FUNCTION_BLOCK FB_QM_MinDirChanges IMPLEMENTS IF_queueManager
VAR_INPUT
	bButtons 	  : ARRAY [1..NUMLEVELS] OF BOOL;						(* user input *)
END_VAR
VAR_OUTPUT
END_VAR
VAR
	tPushDetects  : ARRAY [1..NUMLEVELS] OF FB_BinaryInp;				(* FBs to buffer user inputs until being processed *)
	queueManip	  : FB_ArrManip;										(* FB for array manipulation, like sorting etc. *)
	k			  : INT;												(* loop variable *)
	eDirection    : LiftMovingDirection := LiftMovingDirection.up;		(* local variable for moving direction *)
	
	nCurLevel	  : INT(1..NUMLEVELS);									(* current lift position *)
	nQueue		  : ARRAY [1..NUMLEVELS] OF INT;						(* queue, saving next targets in current moving direction *)
	bLevelInQueue : ARRAY [1..NUMLEVELS] OF BOOL;						(* buffer of all active calls , i.e. levels in nQueue OR active tPushDetects *)
END_VAR

FOR k:=1 TO NUMLEVELS DO
	tPushDetects[k](bPush:=bButtons[k], bReset:=FALSE);
	bLevelInQueue[k] := tPushDetects[k].bOutActive OR queueManip.isElement(arr:=nQueue, entry:=k);
END_FOR

FOR k:=1 TO NUMLEVELS DO
	IF tPushDetects[k].bOutActive THEN
		IF queueManip.isEmpty(arr:=nQueue, emptyElement:=0) THEN
			// Queue is empty. Just inset new element and sort desc (-> new Element is at front)
			queueManip.insert(arr:=nQueue, newElement:=k, freeElement:=0);
			queueManip.quicksort_desc(arr:=nQueue, lo:=1, hi:=NUMLEVELS);
			// ... and set Direction to UP if current lift position is below the calling level
			IF nCurLevel < k THEN
				eDirection := LiftMovingDirection.up;
			END_IF
			// ... and set Direction to DOWN if current lift position is above the calling level
			IF nCurLevel > k THEN
				eDirection := LiftMovingDirection.down;
			END_IF
			// otherwise leave direction as it is!
			
			// Then acknowledge
			tPushDetects[k](bReset:=TRUE);
			CONTINUE;
		END_IF	
	
		(*
			if new call is already included in queue, then acknowldge
			and continue with next loop iteration 
		*)
		IF queueManip.isElement(arr:=nQueue, entry:=k) THEN
			tPushDetects[k](bReset:=TRUE);
			CONTINUE;
		END_IF
		
		(* 
			lift is moving up and new call is from above the lift position,
			so the new call in inserted into queue and queue is sorted afterwards.
		*)
		IF nCurLevel < k AND eDirection = LiftMovingDirection.up THEN
			queueManip.insert(arr:=nQueue, newElement:=k, freeElement:=0);
			queueManip.quicksort_asc(arr:=nQueue, lo:=1, hi:=NUMLEVELS);
			WHILE nQueue[1] = 0 DO
				queueManip.pop_front(arr:=nQueue, fill:=0);
			END_WHILE
			// ack call
			tPushDetects[k](bReset:=TRUE);
		END_IF
		
		(* 
			lift is moving down and new call is from below the lift position,
			so the new call in inserted into queue and queue is sorted afterwards.
		*)
		IF nCurLevel > k AND eDirection = LiftMovingDirection.down THEN
			queueManip.insert(arr:=nQueue, newElement:=k, freeElement:=0);
			queueManip.quicksort_desc(arr:=nQueue, lo:=1, hi:=NUMLEVELS);
			// ack call
			tPushDetects[k](bReset:=TRUE);
		END_IF
	END_IF
END_FOR

PROPERTY currentLevel : INT (1..NUMLEVELS)
SET
nCurLevel := currentLevel;
END_SET
END_PROPERTY

METHOD doneAck
VAR_INPUT
END_VAR
VAR
END_VAR
(* 
By calling this method, the first entry in nQueue is deleted and all remaining entries are shiftetd one position forward. 
Method shall be called, after the latest moving job has been executed. 
*)
queueManip.pop_front(arr:=nQueue, fill:=0);
END_METHOD

PROPERTY queue : REFERENCE TO ARRAY [1..NUMLEVELS] OF INT
GET
queue REF= nQueue;
END_GET
END_PROPERTY

METHOD reset
VAR_INPUT
END_VAR
VAR
	i : INT;
END_VAR
(* resets all calls *)
FOR i:=1 TO NUMLEVELS DO
	nQueue[i] := 0;
	tPushDetects[i](bReset:=TRUE);
END_FOR
END_METHOD

END_FUNCTION_BLOCK

(* stored: Version 1.1.0.1, ProductVersion 3.1.4024.6
   POU FB_QM_MinDirChanges: Id {2a7de36e-768f-4ee0-9272-f4d3c2690c2b}, SpecialFunc None
   Property currentLevel: Id {f0e23ccc-d1cd-4859-ba89-89f97026054e}
   Set Set: Id {bfa1cb56-20d0-4330-8d8a-80bb22abfcb5}
   Method doneAck: Id {21a29943-5900-4538-ac43-f748175fb01f}
   Property queue: Id {1215a89b-1f63-430a-b88d-e06ced1b7c72}
   Get Get: Id {bf3bf46a-d03c-44af-8541-3868ad94a145}
   Method reset: Id {c38562d4-0543-4007-9b4e-af4bc26bb9c2} *)
